FUNCTION F_HeaderErrorMessage : STRING
VAR_INPUT
	ErrorID		: UDINT;
END_VAR

IF ErrorID = 0 THEN
	F_HeaderErrorMessage := 'None';
ELSIF ErrorID = 1 THEN
	F_HeaderErrorMessage := 'Startup safety';
END_IF

END_FUNCTION

(* stored: Version 1.1.0.1, ProductVersion 3.1.4024.9
   POU F_HeaderErrorMessage: Id {43c8eb4b-e9ef-4cd2-bfcc-280bd910c30e}, SpecialFunc None *)
